// TIA Portal V19 export
TYPE "LUC_typeEmFeedback"
// stored: Access Published
   STRUCT
      isLinked : Bool := true;   // EM is linked to the parent (usually the unit)
      commands : "LUC_typeStateCommands";
   END_STRUCT;
END_TYPE
